# EPICS substitutions: apps/jscalerApp/Db/jscalers_wf_S2.substitutions
file "db/jscalers_wf_averages-1type-1sector.db" {
pattern { T S }
{ FADC 2 }
{ TRG 2 }
{ TDC 2 }
}
